FUNCTION_BLOCK Motor
VAR_INPUT
	MotorInputs : MotorInputVariables;
END_VAR
VAR_OUTPUT
	MotorOutputs : MotorOutputVariables;
END_VAR
VAR
	Start : BOOL;
	Stop : BOOL;
END_VAR

Start := MotorInputs.start;
Stop := MotorInputs.stop;
IF Start AND NOT Stop AND NOT MotorInputs.overload THEN
	MotorOutputs.coil := TRUE;
ELSE
	MotorOutputs.coil := FALSE;
END_IF

END_FUNCTION_BLOCK

(* stored: Version 1.1.0.1, ProductVersion 3.1.4024.12
   POU Motor: Id {8e1e9767-7348-4992-838e-044a25fffec2}, SpecialFunc None *)
